// TIA Portal V20 export
FUNCTION_BLOCK "Simulation"   // FB32843, LAD
// stored: MemoryReserve 100, Namespace Unit1.Em11, SetENOAutomatically false
   VAR_INPUT
      simulation { ExternalAccessible := 'False'; ExternalVisible := 'False'; ExternalWritable := 'False'} : Bool;
   END_VAR
   VAR
      statDigitalSignal { ExternalAccessible := 'False'; ExternalVisible := 'False'; ExternalWritable := 'False'} : Array[0..9] of Bool;
   END_VAR
BEGIN

REGION Network 1: Digital Signal
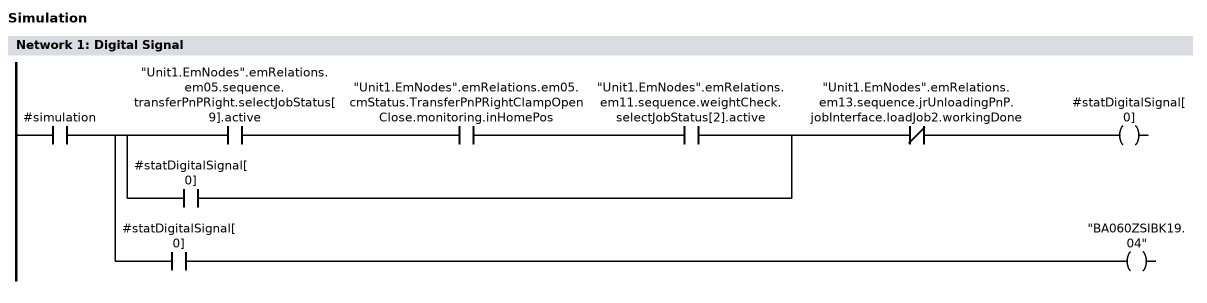
   RUNG wire#powerrail
      Contact( #simulation )
      wire#w1
      Contact( "Unit1.EmNodes".emRelations.em05.sequence.transferPnPRight.selectJobStatus[9].active )
      Contact( "Unit1.EmNodes".emRelations.em05.cmStatus.TransferPnPRightClampOpenClose.monitoring.inHomePos )
      Contact( "Unit1.EmNodes".emRelations.em11.sequence.weightCheck.selectJobStatus[2].active )
      wire#w2
      I_Contact( "Unit1.EmNodes".emRelations.em13.sequence.jrUnloadingPnP.jobInterface.loadJob2.workingDone )
      Coil( #statDigitalSignal[0] )
   END_RUNG
   RUNG wire#w1
      Contact( #statDigitalSignal[0] )
   END_RUNG wire#w2
   RUNG wire#w1
      Contact( #statDigitalSignal[0] )
      Coil( "BA060ZSIBK19.04" )
   END_RUNG
   // the same network as SCL:
   #statDigitalSignal[0] := #simulation AND (("Unit1.EmNodes".emRelations.em05.sequence.transferPnPRight.selectJobStatus[9].active AND "Unit1.EmNodes".emRelations.em05.cmStatus.TransferPnPRightClampOpenClose.monitoring.inHomePos AND "Unit1.EmNodes".emRelations.em11.sequence.weightCheck.selectJobStatus[2].active) OR #statDigitalSignal[0]) AND NOT "Unit1.EmNodes".emRelations.em13.sequence.jrUnloadingPnP.jobInterface.loadJob2.workingDone;
   "BA060ZSIBK19.04" := #simulation AND #statDigitalSignal[0];
END_REGION
END_FUNCTION_BLOCK
